// TIA Portal V18 export
FUNCTION "SS1_710A1_8RTD_IO_Update" : Void   // FC11020, LAD
{ S7_Optimized_Access := 'TRUE' }
VERSION : 0.1
// stored: AutoNumber false, IsIECCheckEnabled false, SetENOAutomatically false, UDAEnableTagReadback false
BEGIN

REGION Network 1
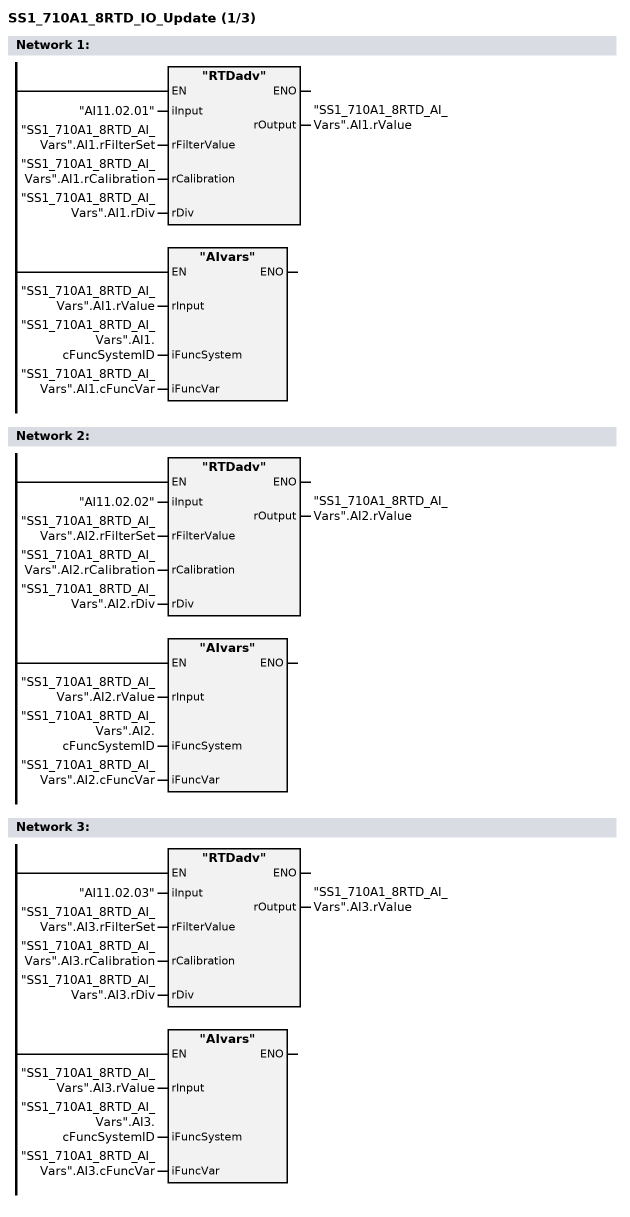
   RUNG wire#powerrail
      "RTDadv"(iInput := "AI11.02.01", rFilterValue := "SS1_710A1_8RTD_AI_Vars".AI1.rFilterSet, rCalibration := "SS1_710A1_8RTD_AI_Vars".AI1.rCalibration, rDiv := "SS1_710A1_8RTD_AI_Vars".AI1.rDiv, rOutput => "SS1_710A1_8RTD_AI_Vars".AI1.rValue)
   END_RUNG
   RUNG wire#powerrail
      "AIvars"(rInput := "SS1_710A1_8RTD_AI_Vars".AI1.rValue, iFuncSystem := "SS1_710A1_8RTD_AI_Vars".AI1.cFuncSystemID, iFuncVar := "SS1_710A1_8RTD_AI_Vars".AI1.cFuncVar)
   END_RUNG
   // the same network as SCL:
   "RTDadv"(iInput := "AI11.02.01",
            rFilterValue := "SS1_710A1_8RTD_AI_Vars".AI1.rFilterSet,
            rCalibration := "SS1_710A1_8RTD_AI_Vars".AI1.rCalibration,
            rDiv := "SS1_710A1_8RTD_AI_Vars".AI1.rDiv,
            rOutput => "SS1_710A1_8RTD_AI_Vars".AI1.rValue);
   "AIvars"(rInput := "SS1_710A1_8RTD_AI_Vars".AI1.rValue,
            iFuncSystem := "SS1_710A1_8RTD_AI_Vars".AI1.cFuncSystemID,
            iFuncVar := "SS1_710A1_8RTD_AI_Vars".AI1.cFuncVar);
END_REGION

REGION Network 2
   RUNG wire#powerrail
      "RTDadv"(iInput := "AI11.02.02", rFilterValue := "SS1_710A1_8RTD_AI_Vars".AI2.rFilterSet, rCalibration := "SS1_710A1_8RTD_AI_Vars".AI2.rCalibration, rDiv := "SS1_710A1_8RTD_AI_Vars".AI2.rDiv, rOutput => "SS1_710A1_8RTD_AI_Vars".AI2.rValue)
   END_RUNG
   RUNG wire#powerrail
      "AIvars"(rInput := "SS1_710A1_8RTD_AI_Vars".AI2.rValue, iFuncSystem := "SS1_710A1_8RTD_AI_Vars".AI2.cFuncSystemID, iFuncVar := "SS1_710A1_8RTD_AI_Vars".AI2.cFuncVar)
   END_RUNG
   // the same network as SCL:
   "RTDadv"(iInput := "AI11.02.02",
            rFilterValue := "SS1_710A1_8RTD_AI_Vars".AI2.rFilterSet,
            rCalibration := "SS1_710A1_8RTD_AI_Vars".AI2.rCalibration,
            rDiv := "SS1_710A1_8RTD_AI_Vars".AI2.rDiv,
            rOutput => "SS1_710A1_8RTD_AI_Vars".AI2.rValue);
   "AIvars"(rInput := "SS1_710A1_8RTD_AI_Vars".AI2.rValue,
            iFuncSystem := "SS1_710A1_8RTD_AI_Vars".AI2.cFuncSystemID,
            iFuncVar := "SS1_710A1_8RTD_AI_Vars".AI2.cFuncVar);
END_REGION

REGION Network 3
   RUNG wire#powerrail
      "RTDadv"(iInput := "AI11.02.03", rFilterValue := "SS1_710A1_8RTD_AI_Vars".AI3.rFilterSet, rCalibration := "SS1_710A1_8RTD_AI_Vars".AI3.rCalibration, rDiv := "SS1_710A1_8RTD_AI_Vars".AI3.rDiv, rOutput => "SS1_710A1_8RTD_AI_Vars".AI3.rValue)
   END_RUNG
   RUNG wire#powerrail
      "AIvars"(rInput := "SS1_710A1_8RTD_AI_Vars".AI3.rValue, iFuncSystem := "SS1_710A1_8RTD_AI_Vars".AI3.cFuncSystemID, iFuncVar := "SS1_710A1_8RTD_AI_Vars".AI3.cFuncVar)
   END_RUNG
   // the same network as SCL:
   "RTDadv"(iInput := "AI11.02.03",
            rFilterValue := "SS1_710A1_8RTD_AI_Vars".AI3.rFilterSet,
            rCalibration := "SS1_710A1_8RTD_AI_Vars".AI3.rCalibration,
            rDiv := "SS1_710A1_8RTD_AI_Vars".AI3.rDiv,
            rOutput => "SS1_710A1_8RTD_AI_Vars".AI3.rValue);
   "AIvars"(rInput := "SS1_710A1_8RTD_AI_Vars".AI3.rValue,
            iFuncSystem := "SS1_710A1_8RTD_AI_Vars".AI3.cFuncSystemID,
            iFuncVar := "SS1_710A1_8RTD_AI_Vars".AI3.cFuncVar);
END_REGION

REGION Network 4
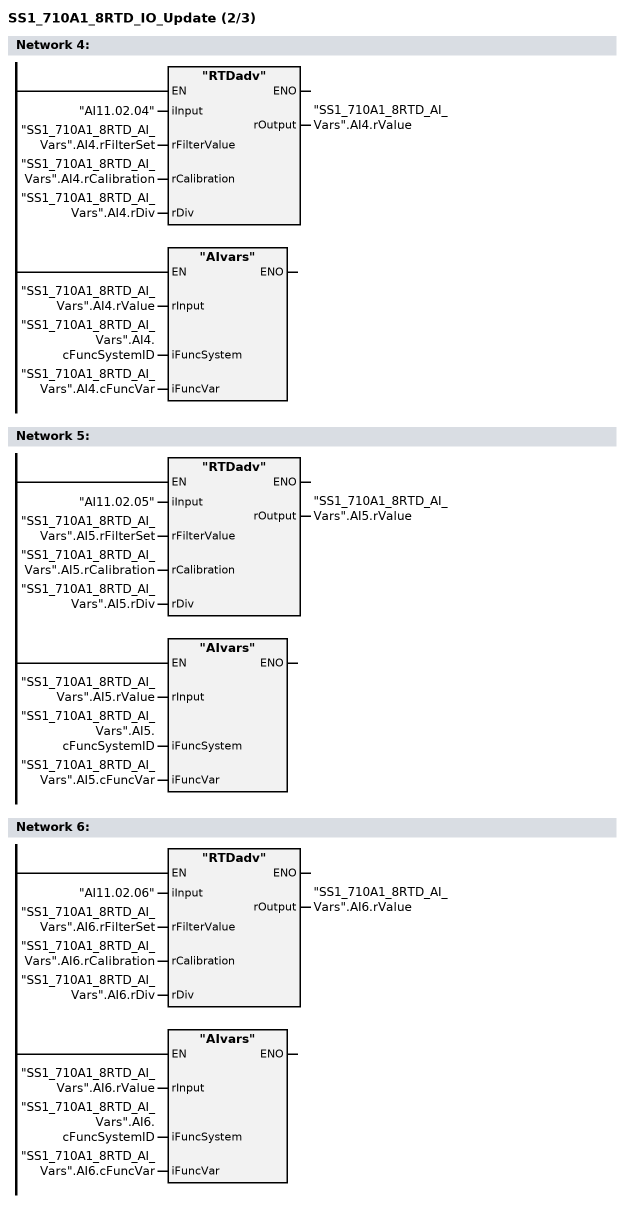
   RUNG wire#powerrail
      "RTDadv"(iInput := "AI11.02.04", rFilterValue := "SS1_710A1_8RTD_AI_Vars".AI4.rFilterSet, rCalibration := "SS1_710A1_8RTD_AI_Vars".AI4.rCalibration, rDiv := "SS1_710A1_8RTD_AI_Vars".AI4.rDiv, rOutput => "SS1_710A1_8RTD_AI_Vars".AI4.rValue)
   END_RUNG
   RUNG wire#powerrail
      "AIvars"(rInput := "SS1_710A1_8RTD_AI_Vars".AI4.rValue, iFuncSystem := "SS1_710A1_8RTD_AI_Vars".AI4.cFuncSystemID, iFuncVar := "SS1_710A1_8RTD_AI_Vars".AI4.cFuncVar)
   END_RUNG
   // the same network as SCL:
   "RTDadv"(iInput := "AI11.02.04",
            rFilterValue := "SS1_710A1_8RTD_AI_Vars".AI4.rFilterSet,
            rCalibration := "SS1_710A1_8RTD_AI_Vars".AI4.rCalibration,
            rDiv := "SS1_710A1_8RTD_AI_Vars".AI4.rDiv,
            rOutput => "SS1_710A1_8RTD_AI_Vars".AI4.rValue);
   "AIvars"(rInput := "SS1_710A1_8RTD_AI_Vars".AI4.rValue,
            iFuncSystem := "SS1_710A1_8RTD_AI_Vars".AI4.cFuncSystemID,
            iFuncVar := "SS1_710A1_8RTD_AI_Vars".AI4.cFuncVar);
END_REGION

REGION Network 5
   RUNG wire#powerrail
      "RTDadv"(iInput := "AI11.02.05", rFilterValue := "SS1_710A1_8RTD_AI_Vars".AI5.rFilterSet, rCalibration := "SS1_710A1_8RTD_AI_Vars".AI5.rCalibration, rDiv := "SS1_710A1_8RTD_AI_Vars".AI5.rDiv, rOutput => "SS1_710A1_8RTD_AI_Vars".AI5.rValue)
   END_RUNG
   RUNG wire#powerrail
      "AIvars"(rInput := "SS1_710A1_8RTD_AI_Vars".AI5.rValue, iFuncSystem := "SS1_710A1_8RTD_AI_Vars".AI5.cFuncSystemID, iFuncVar := "SS1_710A1_8RTD_AI_Vars".AI5.cFuncVar)
   END_RUNG
   // the same network as SCL:
   "RTDadv"(iInput := "AI11.02.05",
            rFilterValue := "SS1_710A1_8RTD_AI_Vars".AI5.rFilterSet,
            rCalibration := "SS1_710A1_8RTD_AI_Vars".AI5.rCalibration,
            rDiv := "SS1_710A1_8RTD_AI_Vars".AI5.rDiv,
            rOutput => "SS1_710A1_8RTD_AI_Vars".AI5.rValue);
   "AIvars"(rInput := "SS1_710A1_8RTD_AI_Vars".AI5.rValue,
            iFuncSystem := "SS1_710A1_8RTD_AI_Vars".AI5.cFuncSystemID,
            iFuncVar := "SS1_710A1_8RTD_AI_Vars".AI5.cFuncVar);
END_REGION

REGION Network 6
   RUNG wire#powerrail
      "RTDadv"(iInput := "AI11.02.06", rFilterValue := "SS1_710A1_8RTD_AI_Vars".AI6.rFilterSet, rCalibration := "SS1_710A1_8RTD_AI_Vars".AI6.rCalibration, rDiv := "SS1_710A1_8RTD_AI_Vars".AI6.rDiv, rOutput => "SS1_710A1_8RTD_AI_Vars".AI6.rValue)
   END_RUNG
   RUNG wire#powerrail
      "AIvars"(rInput := "SS1_710A1_8RTD_AI_Vars".AI6.rValue, iFuncSystem := "SS1_710A1_8RTD_AI_Vars".AI6.cFuncSystemID, iFuncVar := "SS1_710A1_8RTD_AI_Vars".AI6.cFuncVar)
   END_RUNG
   // the same network as SCL:
   "RTDadv"(iInput := "AI11.02.06",
            rFilterValue := "SS1_710A1_8RTD_AI_Vars".AI6.rFilterSet,
            rCalibration := "SS1_710A1_8RTD_AI_Vars".AI6.rCalibration,
            rDiv := "SS1_710A1_8RTD_AI_Vars".AI6.rDiv,
            rOutput => "SS1_710A1_8RTD_AI_Vars".AI6.rValue);
   "AIvars"(rInput := "SS1_710A1_8RTD_AI_Vars".AI6.rValue,
            iFuncSystem := "SS1_710A1_8RTD_AI_Vars".AI6.cFuncSystemID,
            iFuncVar := "SS1_710A1_8RTD_AI_Vars".AI6.cFuncVar);
END_REGION

REGION Network 7
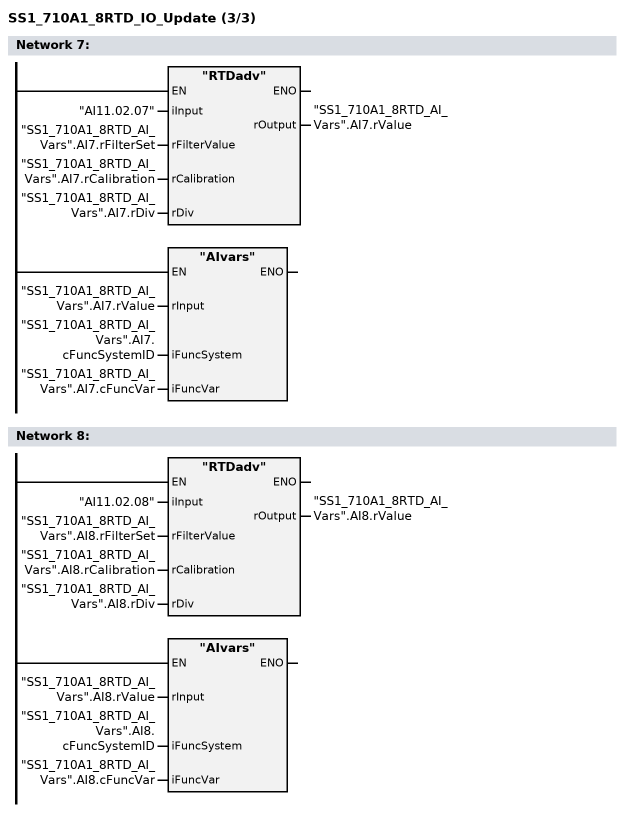
   RUNG wire#powerrail
      "RTDadv"(iInput := "AI11.02.07", rFilterValue := "SS1_710A1_8RTD_AI_Vars".AI7.rFilterSet, rCalibration := "SS1_710A1_8RTD_AI_Vars".AI7.rCalibration, rDiv := "SS1_710A1_8RTD_AI_Vars".AI7.rDiv, rOutput => "SS1_710A1_8RTD_AI_Vars".AI7.rValue)
   END_RUNG
   RUNG wire#powerrail
      "AIvars"(rInput := "SS1_710A1_8RTD_AI_Vars".AI7.rValue, iFuncSystem := "SS1_710A1_8RTD_AI_Vars".AI7.cFuncSystemID, iFuncVar := "SS1_710A1_8RTD_AI_Vars".AI7.cFuncVar)
   END_RUNG
   // the same network as SCL:
   "RTDadv"(iInput := "AI11.02.07",
            rFilterValue := "SS1_710A1_8RTD_AI_Vars".AI7.rFilterSet,
            rCalibration := "SS1_710A1_8RTD_AI_Vars".AI7.rCalibration,
            rDiv := "SS1_710A1_8RTD_AI_Vars".AI7.rDiv,
            rOutput => "SS1_710A1_8RTD_AI_Vars".AI7.rValue);
   "AIvars"(rInput := "SS1_710A1_8RTD_AI_Vars".AI7.rValue,
            iFuncSystem := "SS1_710A1_8RTD_AI_Vars".AI7.cFuncSystemID,
            iFuncVar := "SS1_710A1_8RTD_AI_Vars".AI7.cFuncVar);
END_REGION

REGION Network 8
   RUNG wire#powerrail
      "RTDadv"(iInput := "AI11.02.08", rFilterValue := "SS1_710A1_8RTD_AI_Vars".AI8.rFilterSet, rCalibration := "SS1_710A1_8RTD_AI_Vars".AI8.rCalibration, rDiv := "SS1_710A1_8RTD_AI_Vars".AI8.rDiv, rOutput => "SS1_710A1_8RTD_AI_Vars".AI8.rValue)
   END_RUNG
   RUNG wire#powerrail
      "AIvars"(rInput := "SS1_710A1_8RTD_AI_Vars".AI8.rValue, iFuncSystem := "SS1_710A1_8RTD_AI_Vars".AI8.cFuncSystemID, iFuncVar := "SS1_710A1_8RTD_AI_Vars".AI8.cFuncVar)
   END_RUNG
   // the same network as SCL:
   "RTDadv"(iInput := "AI11.02.08",
            rFilterValue := "SS1_710A1_8RTD_AI_Vars".AI8.rFilterSet,
            rCalibration := "SS1_710A1_8RTD_AI_Vars".AI8.rCalibration,
            rDiv := "SS1_710A1_8RTD_AI_Vars".AI8.rDiv,
            rOutput => "SS1_710A1_8RTD_AI_Vars".AI8.rValue);
   "AIvars"(rInput := "SS1_710A1_8RTD_AI_Vars".AI8.rValue,
            iFuncSystem := "SS1_710A1_8RTD_AI_Vars".AI8.cFuncSystemID,
            iFuncVar := "SS1_710A1_8RTD_AI_Vars".AI8.cFuncVar);
END_REGION
END_FUNCTION
